PROGRAM OP10_MANUAL
VAR
//OP10A
	OP10A_O_HORZ_MANUALPB1							: BOOL;
	OP10A_O_HORZ_MANUALPB2							: BOOL;
	OP10A_O_VERT_MANUALPB1							: BOOL;
	OP10A_O_VERT_MANUALPB2							: BOOL;
	OP10A_M_O_LHGRIP_ONOFF							: BOOL;
	OP10A_M_O_RHGRIP_ONOFF							: BOOL;
	OP10A_M_O_LHPUSH_CYL							: BOOL;
	OP10A_M_O_RHPUSH_CYL							: BOOL;	
	OP10A_O_0DEGRE_MANUALPB1						: BOOL;
	OP10A_O_180DEGRE_MANUALPB2						: BOOL;
	OP10A_M_LNR1_ONOFF								: BOOL;
	OP10A_M_LNR2_ONOFF								: BOOL;
	OP10A_M_BOWL_ONOFF								: BOOL;
	OP10A_M_HOPPER_ONOFF							: BOOL;
	OP10A_M_LH_REJ_WRK								: BOOL;
	OP10A_M_LH_REJ_HOME								: BOOL;
	OP10A_M_RH_REJ_HOME								: BOOL;
	OP10A_M_RH_REJ_WRK								: BOOL;
	OP10_FRT_BDY_SING_HME							: BOOL;
	OP10_FRT_BDY_SING_WRK							: BOOL;	
	OP10_SEC_BDY_SING_HME							: BOOL;
	OP10_SEC_BDY_SING_WRK							: BOOL;	
	
	
//OP10B                                     		
	OP10B_O_HORZ_MANUALPB1							: BOOL;
	OP10B_O_HORZ_MANUALPB2							: BOOL;
	OP10B_O_VERT_MANUALPB1							: BOOL;
	OP10B_O_VERT_MANUALPB2							: BOOL;
	OP10B_M_O_LHGRIP_ONOFF							: BOOL;
	OP10B_M_O_RHGRIP_ONOFF							: BOOL;
	OP10B_M_O_LHPUSH_CYL							: BOOL;
	OP10B_M_O_RHPUSH_CYL							: BOOL;
	OP10B_O_0DEGRE_MANUALPB1						: BOOL;
	OP10B_O_180DEGRE_MANUALPB2						: BOOL;
	OP10B_M_LNR1_ONOFF								: BOOL;
	OP10B_M_LNR2_ONOFF								: BOOL;
	OP10B_M_BOWL_ONOFF								: BOOL;
	OP10B_M_HOPPER_ONOFF							: BOOL;
	OP10B_M_LH_REJ_HOME								: BOOL;
	OP10B_M_LH_REJ_WRK								: BOOL;
	OP10B_M_RH_REJ_HOME								: BOOL;
	OP10B_M_RH_REJ_WRK								: BOOL;
	
// ALARM BITS

	OP10A_HORZ_CYL_A1								: BOOL;
	OP10A_HORZ_CYL_A2								: BOOL;
	OP10A_HORZ_CYL_A3								: BOOL;
	OP10A_HORZ_CYL_A4								: BOOL;
	OP10A_HORZ_CYL_A5								: BOOL;
	OP10A_VERT_CYL_A1								: BOOL;
	OP10A_VERT_CYL_A2								: BOOL;
	OP10A_VERT_CYL_A3								: BOOL;
	OP10A_VERT_CYL_A4								: BOOL;
	OP10A_VERT_CYL_A5								: BOOL;
	OP10A_DEGREE_CYL_A1								: BOOL;
	OP10A_DEGREE_CYL_A2								: BOOL;
	OP10A_DEGREE_CYL_A3								: BOOL;
	OP10A_DEGREE_CYL_A4								: BOOL;
	OP10A_DEGREE_CYL_A5								: BOOL;
	OP10A_LH_GRP_A1									: BOOL;
	OP10A_LH_GRP_A2									: BOOL;
	OP10A_LH_GRP_A3									: BOOL;
	OP10A_LH_GRP_A4									: BOOL;
	OP10A_LH_GRP_A5									: BOOL;
	OP10A_RH_GRP_A1									: BOOL;
	OP10A_RH_GRP_A2									: BOOL;
	OP10A_RH_GRP_A3									: BOOL;
	OP10A_RH_GRP_A4									: BOOL;
	OP10A_RH_GRP_A5									: BOOL;
	OP10A_LH_PUSH_A1								: BOOL;
	OP10A_LH_PUSH_A2								: BOOL;
	OP10A_LH_PUSH_A3								: BOOL;
	OP10A_LH_PUSH_A4								: BOOL;
	OP10A_LH_PUSH_A5								: BOOL;
	OP10A_RH_PUSH_A1								: BOOL;
	OP10A_RH_PUSH_A2								: BOOL;
	OP10A_RH_PUSH_A3								: BOOL;
	OP10A_RH_PUSH_A4								: BOOL;
	OP10A_RH_PUSH_A5								: BOOL;
	OP10A_LH_REJ_A1									: BOOL;
	OP10A_LH_REJ_A2									: BOOL;
	OP10A_LH_REJ_A3									: BOOL;
	OP10A_LH_REJ_A4									: BOOL;
	OP10A_LH_REJ_A5									: BOOL;
	OP10A_RH_REJ_A1									: BOOL;
	OP10A_RH_REJ_A2									: BOOL;
	OP10A_RH_REJ_A3									: BOOL;
	OP10A_RH_REJ_A4									: BOOL;
	OP10A_RH_REJ_A5									: BOOL;
	OP10B_HORZ_CYL_A1								: BOOL;
	OP10B_HORZ_CYL_A2								: BOOL;
	OP10B_HORZ_CYL_A3								: BOOL;
	OP10B_HORZ_CYL_A4								: BOOL;
	OP10B_HORZ_CYL_A5								: BOOL;
	OP10B_VERT_CYL_A1								: BOOL;
	OP10B_VERT_CYL_A2								: BOOL;
	OP10B_VERT_CYL_A3								: BOOL;
	OP10B_VERT_CYL_A4								: BOOL;
	OP10B_VERT_CYL_A5								: BOOL;
	OP10B_DEGREE_CYL_A1								: BOOL;
	OP10B_DEGREE_CYL_A2								: BOOL;
	OP10B_DEGREE_CYL_A3								: BOOL;
	OP10B_DEGREE_CYL_A4								: BOOL;
	OP10B_DEGREE_CYL_A5								: BOOL;
	OP10B_LH_GRP_A1									: BOOL;
	OP10B_LH_GRP_A2									: BOOL;
	OP10B_LH_GRP_A3									: BOOL;
	OP10B_LH_GRP_A4									: BOOL;
	OP10B_LH_GRP_A5									: BOOL;
	OP10B_RH_GRP_A1									: BOOL;
	OP10B_RH_GRP_A2									: BOOL;
	OP10B_RH_GRP_A3									: BOOL;
	OP10B_RH_GRP_A4									: BOOL;
	OP10B_RH_GRP_A5									: BOOL;
	OP10B_LH_PUSH_A1								: BOOL;
	OP10B_LH_PUSH_A2								: BOOL;
	OP10B_LH_PUSH_A3								: BOOL;
	OP10B_LH_PUSH_A4								: BOOL;
	OP10B_LH_PUSH_A5								: BOOL;
	OP10B_RH_PUSH_A1								: BOOL;
	OP10B_RH_PUSH_A2								: BOOL;
	OP10B_RH_PUSH_A3								: BOOL;
	OP10B_RH_PUSH_A4								: BOOL;
	OP10B_RH_PUSH_A5								: BOOL;
	OP10B_LH_REJ_A1									: BOOL;
	OP10B_LH_REJ_A2									: BOOL;
	OP10B_LH_REJ_A3									: BOOL;
	OP10B_LH_REJ_A4									: BOOL;
	OP10B_LH_REJ_A5									: BOOL;
	OP10B_RH_REJ_A1									: BOOL;
	OP10B_RH_REJ_A2									: BOOL;
	OP10B_RH_REJ_A3									: BOOL;
	OP10B_RH_REJ_A4									: BOOL;
	OP10B_RH_REJ_A5									: BOOL;	
	OP10_BDY_SING_FRT_A1							: BOOL;
	OP10_BDY_SING_FRT_A2							: BOOL;
	OP10_BDY_SING_FRT_A3							: BOOL;
	OP10_BDY_SING_FRT_A4							: BOOL;
	OP10_BDY_SING_FRT_A5							: BOOL;	
	OP10_BDY_SING_SEC_A1							: BOOL;
	OP10_BDY_SING_SEC_A2							: BOOL;
	OP10_BDY_SING_SEC_A3							: BOOL;
	OP10_BDY_SING_SEC_A4							: BOOL;
	OP10_BDY_SING_SEC_A5							: BOOL;	
	
	
	

//INT

	OP10A_HORZ_CYL_STUS								: INT;
	OP10A_VERT_CYL_STUS								: INT;
	OP10A_DEGREE_CYL_STUS							: INT;
	OP10A_LH_GRP_STATS								: INT;
	OP10A_RH_GRP_STUS								: INT;
	OP10A_LH_PUSH_STUS								: INT;
	OP10A_RH_PUSH_STUS								: INT;
	OP10B_HORZ_CYL_STUS								: INT;
	OP10B_VERT_CYL_STUS								: INT;
	OP10B_DEGREE_CYL_STUS							: INT;
	OP10B_LH_GRP_STATS								: INT;
	OP10B_RH_GRP_STUS								: INT;
	OP10B_LH_PUSH_STUS								: INT;
	OP10B_RH_PUSH_STUS								: INT;
                              				
// BOOL                             				
	OP10A_H_LNR1_ONOFF								: BOOL;
	OP10A_H_LNR2_ONOFF								: BOOL;
	OP10A_H_BOWL_ONOFF								: BOOL;
	OP10A_H_HOPPER_ONOFF							: BOOL;
	OP10B_H_LNR1_ONOFF								: BOOL;
	OP10B_H_LNR2_ONOFF								: BOOL;
	OP10B_H_BOWL_ONOFF								: BOOL;
	OP10B_H_HOPPER_ONOFF							: BOOL;

	
	
	
HMI_TRIAL_SWITH_GOKUL_2							:BOOL;	
	
TEMP	: BOOL;
	temp1: BOOL;
	temp2: BOOL;
	OP10_BDY_SING_FRT_STATUS: INT;
	OP10_BDY_SING_SEC_STATUS: INT;




	OP10B_PARLLEL: INT;
	OP10A_PARALLEL: INT;
END_VAR

VAR RETAIN

END_VAR

//#############################		OP10A		###############################

IF OP10A_MANUAL_SELECTED THEN

//OP10A
	OP10A_M_LNR1_ONOFF							:= OP10A_H_LNR1_ONOFF;
	OP10A_M_LNR2_ONOFF          				:= OP10A_H_LNR2_ONOFF;
	OP10A_M_BOWL_ONOFF          				:= OP10A_H_BOWL_ONOFF;
	OP10A_M_HOPPER_ONOFF        				:= OP10A_H_HOPPER_ONOFF;	

CASE OP10_CYL_NO OF                 		
	                                		
	1: IF OP10_HOME THEN            		
		OP10A_O_HORZ_MANUALPB1					:=TRUE;
		OP10A_O_HORZ_MANUALPB2					:=FALSE;
		END_IF                      			
		IF OP10_WORK THEN           			
		OP10A_O_HORZ_MANUALPB1					:=FALSE;
		OP10A_O_HORZ_MANUALPB2					:=TRUE;
		END_IF                      			
                                    			
	2: IF OP10_HOME THEN            			
		OP10A_O_VERT_MANUALPB1					:=TRUE;
		OP10A_O_VERT_MANUALPB2					:=FALSE;
		END_IF                      		
		IF OP10_WORK THEN           		
		OP10A_O_VERT_MANUALPB1					:=FALSE;
		OP10A_O_VERT_MANUALPB2					:=TRUE;
		END_IF                      			
		                            			
	4:IF OP10_HOME THEN             			
		OP10A_O_0DEGRE_MANUALPB1				:=TRUE;
		OP10A_O_180DEGRE_MANUALPB2				:=FALSE;
		END_IF                      			
		IF OP10_WORK THEN           			
		OP10A_O_0DEGRE_MANUALPB1				:=FALSE;
		OP10A_O_180DEGRE_MANUALPB2				:=TRUE;
		END_IF                      		
                            		
	9: IF OP10_HOME THEN            		
		OP10A_M_LH_REJ_HOME						:=TRUE;
		OP10A_M_LH_REJ_WRK		 				:=FALSE;
		END_IF                      			
		IF OP10_WORK THEN           			
		OP10A_M_LH_REJ_HOME						:=FALSE;
		OP10A_M_LH_REJ_WRK	 					:=TRUE;
		END_IF                      			
		                            			
	10: IF OP10_HOME THEN           			
		OP10A_M_RH_REJ_HOME						:=TRUE;
		OP10A_M_RH_REJ_WRK	 	 				:=FALSE;
		END_IF                      			
		IF OP10_WORK THEN           			
		OP10A_M_RH_REJ_HOME						:=FALSE;
		OP10A_M_RH_REJ_WRK	 					:=TRUE;
		END_IF	                    		
		                            		                     		
		                            		
	13: IF OP10_HOME THEN           		
		OP10A_M_O_LHGRIP_ONOFF					:=FALSE;
		END_IF                      			
		IF OP10_WORK THEN           			
		OP10A_M_O_LHGRIP_ONOFF					:=TRUE;
		END_IF                      			
		                            			
	14:	IF OP10_HOME THEN           			
		OP10A_M_O_RHGRIP_ONOFF					:=FALSE;
		END_IF                      			
		IF OP10_WORK THEN           	    	
		OP10A_M_O_RHGRIP_ONOFF					:=TRUE;
		END_IF                      			
		                            			
	15: IF OP10_HOME THEN           			
		OP10A_M_O_LHPUSH_CYL					:=FALSE;
		END_IF                      		
		IF OP10_WORK THEN           		
		OP10A_M_O_LHPUSH_CYL					:=TRUE;
		END_IF                      			
		                            			
	16: IF OP10_HOME THEN           			
		OP10A_M_O_RHPUSH_CYL					:=FALSE;
		END_IF                      			
		IF OP10_WORK THEN           			
		OP10A_M_O_RHPUSH_CYL					:=TRUE;
		END_IF                              	
		                                    	
	17: IF OP10_HOME THEN           			
		OP10_FRT_BDY_SING_HME					:=TRUE;
		OP10_FRT_BDY_SING_WRK 	 				:=FALSE;
		END_IF                      		
		IF OP10_WORK THEN           		
		OP10_FRT_BDY_SING_HME	 				:=FALSE;
		OP10_FRT_BDY_SING_WRK 					:=TRUE;
		END_IF                              	
                                            	
	18: IF OP10_HOME THEN           			
		OP10_SEC_BDY_SING_HME					:=TRUE;
		OP10_SEC_BDY_SING_WRK		 			:=FALSE;
		END_IF                      		
		IF OP10_WORK THEN           		
		OP10_SEC_BDY_SING_HME					:=FALSE;
		OP10_SEC_BDY_SING_WRK					:=TRUE;
		END_IF                              	
                    		                	
		                            	    	
END_CASE

CASE OP10_SERVO_NO OF               	
	                                	
	1: OP10A_SRV_O_CNVY_STUS.jogPos				:= OP10_JOG_POSITIVE AND NOT OP10_JOG_NEGATIVE;
	   OP10A_SRV_O_CNVY_STUS.jogNeg				:= OP10_JOG_NEGATIVE AND NOT OP10_JOG_POSITIVE;
	   OP10A_SRV_O_CNVY_CNT.Bsethome	        := OP10A_SET_HOME;
	   OP10A_SRV_O_CNVY_STUS.targetPositon	    := OP10A_TARGET_POSITION;
	   OP10A_SRV_O_CNVY_STUS.moveAbsolute	    := OP10A_MOVE_TARGET;
	   OP10A_SRV_ACT_POS						:= OP10A_SRV_O_CNVY_STUS.actualPosition;
	   OP10A_SRV_FAULT							:= OP10A_CONVEYOR.bAxisError;
	   OP10A_SRV_ENABLE							:= OP10A_CONVEYOR.bAxisEnabled;

	    
	3: OP10A_SRV_LH_BDYGRP_STUS.jogPos			:= OP10_JOG_POSITIVE AND NOT OP10_JOG_NEGATIVE;
	   OP10A_SRV_LH_BDYGRP_STUS.jogNeg      	:= OP10_JOG_NEGATIVE AND NOT OP10_JOG_POSITIVE;  
	   OP10A_SRV_LH_BDYGRP_CNT.Axis_Home_Cmd	:= OP10A_SET_HOME;
	   OP10A_SRV_LH_BDYGRP_STUS.targetPositon	:= OP10A_TARGET_POSITION;
	   OP10A_SRV_LH_BDYGRP_STUS.moveAbsolute	:= OP10A_MOVE_TARGET;
	   OP10A_SRV_ACT_POS						:= OP10A_SRV_LH_BDYGRP_STUS.actualPosition;
	   OP10A_SRV_FAULT							:= OP10A_LH_GRIPR.bAxisError;
	   OP10A_SRV_ENABLE							:= OP10A_LH_GRIPR.bAxisEnabled;
	   
	4: OP10A_SRV_RH_BDYGRP_STUS.jogPos			:= OP10_JOG_POSITIVE AND NOT OP10_JOG_NEGATIVE;
	   OP10A_SRV_RH_BDYGRP_STUS.jogNeg   		:= OP10_JOG_NEGATIVE AND NOT OP10_JOG_POSITIVE;
	   OP10A_SRV_RH_BDYGRP_CNT.Axis_Home_Cmd	:= OP10A_SET_HOME;
	   OP10A_SRV_RH_BDYGRP_STUS.targetPositon	:= OP10A_TARGET_POSITION;
	   OP10A_SRV_RH_BDYGRP_STUS.moveAbsolute	:= OP10A_MOVE_TARGET;
	   OP10A_SRV_ACT_POS						:= OP10A_SRV_RH_BDYGRP_STUS.actualPosition;
	   OP10A_SRV_FAULT							:= OP10A_RH_GRIPR.bAxisError;
	   OP10A_SRV_ENABLE							:= OP10A_RH_GRIPR.bAxisEnabled;
	                                			
	5: OP10A_SRV_LH_BDYANG_STUS.jogPos			:= OP10_JOG_POSITIVE AND NOT OP10_JOG_NEGATIVE;
	   OP10A_SRV_LH_BDYANG_STUS.jogNeg   		:= OP10_JOG_NEGATIVE AND NOT OP10_JOG_POSITIVE;
	   OP10A_SRV_LH_BDYANG_CNT.Axis_Home_Cmd	:= OP10A_SET_HOME;
	   OP10A_SRV_LH_BDYANG_STUS.targetPositon	:= OP10A_TARGET_POSITION;
	   OP10A_SRV_LH_BDYANG_STUS.moveAbsolute	:= OP10A_MOVE_TARGET;
	   OP10A_SRV_ACT_POS						:= OP10A_SRV_LH_BDYANG_STUS.actualPosition;
	   OP10A_SRV_FAULT							:= OP10A_LH_ROTY.bAxisError;
	   OP10A_SRV_ENABLE							:= OP10A_LH_ROTY.bAxisEnabled;
                                			
	6: OP10A_SRV_RH_BDYANG_STUS.jogPos			:= OP10_JOG_POSITIVE AND NOT OP10_JOG_NEGATIVE;
	   OP10A_SRV_RH_BDYANG_STUS.jogNeg   		:= OP10_JOG_NEGATIVE AND NOT OP10_JOG_POSITIVE;
	   OP10A_SRV_RH_BDYANG_CNT.Axis_Home_Cmd	:= OP10A_SET_HOME;
	   OP10A_SRV_RH_BDYANG_STUS.targetPositon	:= OP10A_TARGET_POSITION;
	   OP10A_SRV_RH_BDYANG_STUS.moveAbsolute	:= OP10A_MOVE_TARGET;
	   OP10A_SRV_ACT_POS						:= OP10A_SRV_RH_BDYANG_STUS.actualPosition;
	   OP10A_SRV_FAULT							:= OP10A_RH_ROTY.bAxisError;
	   OP10A_SRV_ENABLE							:= OP10A_RH_ROTY.bAxisEnabled;
                           			
	11:OP10_SRV_FRST_PCKBDY_STUS.jogPos			:= OP10_JOG_POSITIVE AND NOT OP10_JOG_NEGATIVE;
	   OP10_SRV_FRST_PCKBDY_STUS.jogNeg  		:= OP10_JOG_NEGATIVE AND NOT OP10_JOG_POSITIVE;
	   OP10_SRV_FRST_PCKBDY_CNT.Axis_Home_Cmd	:= OP10A_SET_HOME;
	   OP10_SRV_FRST_PCKBDY_STUS.targetPositon	:= OP10A_TARGET_POSITION;    
	   OP10_SRV_FRST_PCKBDY_STUS.moveAbsolute	:= OP10A_MOVE_TARGET;
	   OP10A_SRV_ACT_POS						:= OP10_SRV_FRST_PCKBDY_STUS.actualPosition;
	   OP10A_SRV_FAULT							:= OP10_FRT_BDY_GPR.bAxisError;
	   OP10A_SRV_ENABLE							:= OP10_FRT_BDY_GPR.bAxisEnabled;

                         			
	12:OP10_SRV_SCND_PCKBDY_STUS.jogPos			:= OP10_JOG_POSITIVE AND NOT OP10_JOG_NEGATIVE;
	   OP10_SRV_SCND_PCKBDY_STUS.jogNeg  		:= OP10_JOG_NEGATIVE AND NOT OP10_JOG_POSITIVE;   
	   OP10_SRV_SCND_PCKBDY_CNT.Axis_Home_Cmd	:= OP10A_SET_HOME;
	   OP10_SRV_SCND_PCKBDY_STUS.targetPositon	:= OP10A_TARGET_POSITION;
	   OP10_SRV_SCND_PCKBDY_STUS.moveAbsolute	:= OP10A_MOVE_TARGET;
	   OP10A_SRV_ACT_POS						:= OP10_SRV_SCND_PCKBDY_STUS.actualPosition;
	   OP10A_SRV_FAULT							:= OP10_SEC_BDY_GPR.bAxisError;
	   OP10A_SRV_ENABLE							:= OP10_SEC_BDY_GPR.bAxisEnabled;	   
END_CASE

ELSE
		OP10_CYL_NO									:=0;	
		OP10A_O_HORZ_MANUALPB1						:=FALSE;
		OP10A_O_HORZ_MANUALPB2						:=FALSE;
		OP10A_O_VERT_MANUALPB1						:=FALSE;
		OP10A_O_VERT_MANUALPB2						:=FALSE;
		OP10A_M_O_LHGRIP_ONOFF						:=FALSE;
		OP10A_O_0DEGRE_MANUALPB1					:=FALSE;
		OP10A_O_180DEGRE_MANUALPB2					:=FALSE;
		OP10A_M_O_LHPUSH_CYL						:=FALSE;
		OP10A_M_LNR1_ONOFF		    				:=FALSE;
		OP10A_M_LNR2_ONOFF          				:=FALSE;
		OP10A_M_BOWL_ONOFF         					:=FALSE;
		OP10A_M_HOPPER_ONOFF       					:=FALSE;
		OP10A_M_O_RHPUSH_CYL						:=FALSE;	
		OP10A_M_O_RHGRIP_ONOFF						:=FALSE;
		OP10A_M_RH_REJ_HOME							:=FALSE;
		OP10A_M_RH_REJ_WRK	 						:=FALSE;
		OP10A_M_LH_REJ_HOME							:=FALSE;
		OP10A_M_LH_REJ_WRK	 						:=FALSE;		
		OP10_FRT_BDY_SING_HME	 					:=FALSE;
		OP10_FRT_BDY_SING_WRK						:=FALSE;
		OP10_SEC_BDY_SING_HME	 					:=FALSE;
		OP10_SEC_BDY_SING_WRK						:=FALSE;		
		
		
		
END_IF
	

//#############################		OP10B		###############################



IF OP10B_MANUAL_SELECTED THEN
//OP10B                         				
	OP10B_M_LNR1_ONOFF          				:= OP10B_H_LNR1_ONOFF  ;
	OP10B_M_LNR2_ONOFF          				:= OP10B_H_LNR2_ONOFF  ;
	OP10B_M_BOWL_ONOFF          				:= OP10B_H_BOWL_ONOFF  ;
	OP10B_M_HOPPER_ONOFF        				:= OP10B_H_HOPPER_ONOFF;	

CASE OP10B_CYL_NO OF 

5: IF OP10B_HOME THEN            		
		OP10B_O_HORZ_MANUALPB1					:=TRUE;
		OP10B_O_HORZ_MANUALPB2					:=FALSE;
		END_IF                      			
		IF OP10B_WORK THEN           			
		OP10B_O_HORZ_MANUALPB1					:=FALSE;
		OP10B_O_HORZ_MANUALPB2					:=TRUE;
		END_IF                      			
                                    			
	6: IF OP10B_HOME THEN            			
		OP10B_O_VERT_MANUALPB1					:=TRUE;
		OP10B_O_VERT_MANUALPB2					:=FALSE;
		END_IF                      			
		IF OP10B_WORK THEN           			
		OP10B_O_VERT_MANUALPB1					:=FALSE;
		OP10B_O_VERT_MANUALPB2					:=TRUE;
		END_IF                      		
		                            		
	8:IF OP10B_HOME THEN             		
		OP10B_O_0DEGRE_MANUALPB1				:=TRUE;
		OP10B_O_180DEGRE_MANUALPB2				:=FALSE;
		END_IF                      			
		IF OP10B_WORK THEN           			
		OP10B_O_0DEGRE_MANUALPB1				:=FALSE;
		OP10B_O_180DEGRE_MANUALPB2				:=TRUE;
		END_IF                              	
	                                        	
	11: IF OP10B_HOME THEN           			
		OP10B_M_LH_REJ_HOME						:=TRUE;
		OP10B_M_LH_REJ_WRK	 	 				:=FALSE;
		END_IF                      		
		IF OP10B_WORK THEN           		
		OP10B_M_LH_REJ_HOME						:=FALSE;
		OP10B_M_LH_REJ_WRK	 					:=TRUE;
		END_IF                      			
                       			            	
	12: IF OP10B_HOME THEN           			
		OP10B_M_RH_REJ_HOME						:=TRUE;
		OP10B_M_RH_REJ_WRK	  	 				:=FALSE;
		END_IF                      			
		IF OP10B_WORK THEN           			
		OP10B_M_RH_REJ_HOME						:=FALSE;
		OP10B_M_RH_REJ_WRK	 					:=TRUE;
		END_IF 	

	17: IF OP10B_HOME THEN           		
		OP10B_M_O_LHGRIP_ONOFF					:=FALSE;
		END_IF                      			
		IF OP10B_WORK THEN           			
		OP10B_M_O_LHGRIP_ONOFF					:=TRUE;
		END_IF                      			
		                            			
	18:	IF OP10B_HOME THEN           			
		OP10B_M_O_RHGRIP_ONOFF					:=FALSE;
		END_IF                      			
		IF OP10B_WORK THEN           			
		OP10B_M_O_RHGRIP_ONOFF					:=TRUE;
		END_IF                      			
		                            			
	19: IF OP10B_HOME THEN           			
		OP10B_M_O_LHPUSH_CYL					:=FALSE;
		END_IF                      		
		IF OP10B_WORK THEN           		
		OP10B_M_O_LHPUSH_CYL					:=TRUE;
		END_IF                      			
		                            			
	20: IF OP10B_HOME THEN           			
		OP10B_M_O_RHPUSH_CYL					:=FALSE;
		END_IF                      			
		IF OP10B_WORK THEN           			
		OP10B_M_O_RHPUSH_CYL					:=TRUE;
		END_IF 

END_CASE	
	
CASE OP10B_SERVO_NO OF 
	
	2: OP10B_SRV_O_CNVY_STUS.jogPos				:= OP10B_JOG_POSITIVE AND NOT OP10B_JOG_NEGATIVE;
	   OP10B_SRV_O_CNVY_STUS.jogNeg				:= OP10B_JOG_NEGATIVE AND NOT OP10B_JOG_POSITIVE;
	   OP10B_SRV_O_CNVY_CNT.Bsethome	        := OP10B_SET_HOME;
	   OP10B_SRV_O_CNVY_STUS.targetPositon	    := OP10B_TARGET_POSITION;
//	   OP10B_SRV_LH_BDYGRP_STUS.targetVelocity	:= OP10B_TARGET_VEL;
	   OP10B_SRV_O_CNVY_STUS.moveAbsolute	    := OP10B_MOVE_TARGET;
	   OP10B_SRV_ACT_POS						:= OP10B_SRV_O_CNVY_STUS.actualPosition;
	   OP10B_SRV_FAULT							:= OP10B_CONVEYOR.bAxisError;
	   OP10B_SRV_ENABLE							:= OP10B_CONVEYOR.bAxisEnabled;
                                    	
	7: OP10B_SRV_LH_BDYGRP_STUS.jogPos			:= OP10B_JOG_POSITIVE AND NOT OP10B_JOG_NEGATIVE;
	   OP10B_SRV_LH_BDYGRP_STUS.jogNeg			:= OP10B_JOG_NEGATIVE AND NOT OP10B_JOG_POSITIVE;
	   OP10B_SRV_LH_BDYGRP_CNT.Axis_Home_Cmd	:= OP10B_SET_HOME;
	   OP10B_SRV_LH_BDYGRP_STUS.targetPositon	:= OP10B_TARGET_POSITION;
//	   OP10B_SRV_LH_BDYGRP_STUS.targetVelocity	:= OP10B_TARGET_VEL;
	   OP10B_SRV_LH_BDYGRP_STUS.moveAbsolute	:= OP10B_MOVE_TARGET;
	   OP10B_SRV_ACT_POS						:= OP10B_SRV_LH_BDYGRP_STUS.actualPosition;
	   OP10B_SRV_FAULT							:= OP10B_LH_GRIPR.bAxisError;
	   OP10B_SRV_ENABLE							:= OP10B_LH_GRIPR.bAxisEnabled;	   
	   
	                                		
	8: OP10B_SRV_RH_BDYGRP_STUS.jogPos			:= OP10B_JOG_POSITIVE AND NOT OP10B_JOG_NEGATIVE;
	   OP10B_SRV_RH_BDYGRP_STUS.jogNeg    		:= OP10B_JOG_NEGATIVE AND NOT OP10B_JOG_POSITIVE;
	   OP10B_SRV_RH_BDYGRP_CNT.Axis_Home_Cmd	:= OP10B_SET_HOME;
	   OP10B_SRV_RH_BDYGRP_STUS.targetPositon	:= OP10B_TARGET_POSITION;
//	   OP10B_SRV_RH_BDYGRP_STUS.targetVelocity	:= OP10B_TARGET_VEL;
	   OP10B_SRV_RH_BDYGRP_STUS.moveAbsolute	:= OP10B_MOVE_TARGET;
	   OP10B_SRV_ACT_POS						:= OP10B_SRV_RH_BDYGRP_STUS.actualPosition;
	   OP10B_SRV_FAULT							:= OP10B_RH_GRIPR.bAxisError;
	   OP10B_SRV_ENABLE							:= OP10B_RH_GRIPR.bAxisEnabled;	
	   
	                                			
	9: OP10B_SRV_LH_BDYANG_STUS.jogPos			:= OP10B_JOG_POSITIVE AND NOT OP10B_JOG_NEGATIVE;
	   OP10B_SRV_LH_BDYANG_STUS.jogNeg   		:= OP10B_JOG_NEGATIVE AND NOT OP10B_JOG_POSITIVE;
	   OP10B_SRV_LH_BDYANG_CNT.Axis_Home_Cmd	:= OP10B_SET_HOME;
	   OP10B_SRV_LH_BDYANG_STUS.targetPositon	:= OP10B_TARGET_POSITION;
//	   OP10B_SRV_LH_BDYANG_STUS.targetVelocity	:= OP10B_TARGET_VEL;
	   OP10B_SRV_LH_BDYANG_STUS.moveAbsolute	:= OP10B_MOVE_TARGET;
	   OP10B_SRV_ACT_POS						:= OP10B_SRV_LH_BDYANG_STUS.actualPosition;
	   OP10B_SRV_FAULT							:= OP10B_LH_ROTY.bAxisError;
	   OP10B_SRV_ENABLE							:= OP10B_LH_ROTY.bAxisEnabled;	   
	                                			
	10:OP10B_SRV_RH_BDYANG_STUS.jogPos			:= OP10B_JOG_POSITIVE AND NOT OP10B_JOG_NEGATIVE;
	   OP10B_SRV_RH_BDYANG_STUS.jogNeg    		:= OP10B_JOG_NEGATIVE AND NOT OP10B_JOG_POSITIVE;
	   OP10B_SRV_RH_BDYANG_CNT.Axis_Home_Cmd	:= OP10B_SET_HOME;
	   OP10B_SRV_RH_BDYANG_STUS.targetPositon	:= OP10B_TARGET_POSITION;
//	   OP10B_SRV_RH_BDYANG_STUS.targetVelocity	:= OP10B_TARGET_VEL;
	   OP10B_SRV_RH_BDYANG_STUS.moveAbsolute	:= OP10B_MOVE_TARGET;
	   OP10B_SRV_ACT_POS						:= OP10B_SRV_RH_BDYANG_STUS.actualPosition;
	   OP10B_SRV_FAULT							:= OP10B_RH_ROTY.bAxisError;
	   OP10B_SRV_ENABLE							:= OP10B_RH_ROTY.bAxisEnabled;	

END_CASE	

ELSE
	OP10B_O_HORZ_MANUALPB1						:=FALSE;		
	OP10B_O_HORZ_MANUALPB2						:=FALSE;		
	OP10B_O_VERT_MANUALPB1						:=FALSE;		
	OP10B_O_VERT_MANUALPB2						:=FALSE;		
	OP10B_M_O_LHGRIP_ONOFF						:=FALSE;		
	OP10B_O_0DEGRE_MANUALPB1					:=FALSE;	
	OP10B_O_180DEGRE_MANUALPB2					:=FALSE;
	OP10B_M_O_LHPUSH_CYL  						:=FALSE;		
	OP10B_M_LNR1_ONOFF  						:=FALSE;		
	OP10B_M_LNR2_ONOFF  						:=FALSE;		
	OP10B_M_BOWL_ONOFF  						:=FALSE;		
	OP10B_M_O_RHPUSH_CYL						:=FALSE;
	OP10B_M_O_RHGRIP_ONOFF						:=FALSE;	
	OP10B_M_RH_REJ_HOME							:=FALSE;
	OP10B_M_RH_REJ_WRK	  	 					:=FALSE;	
	OP10B_M_LH_REJ_HOME							:=FALSE;
	OP10B_M_LH_REJ_WRK	 						:=FALSE;

END_IF
// OP10B_HORZ_CYLINDER_SAFE_WRK/HME
OP10A_HORZ_CYL.SafeHome				:=OP10A_VERT_CYL.Sensor1 ;//AND OP10A_DEGREE_CYL.Sensor1;
OP10A_HORZ_CYL.SafeWork             :=OP10A_VERT_CYL.Sensor1 ;//AND OP10A_DEGREE_CYL.Sensor1;


OP10A_HORZ_CYL(
	Auto:= OP10A_AUTO_RUNNING OR OP10A_STEP_RUNNING OR OP10A_CYL_PNP_CHECK, 
	Manual:= OP10A_MANUAL_SELECTED,
	HOMING_RUNNING:= OP10A_START_HOMNG, 
	ErrorActive:= OP10A_ERR, 
	ResetPB:= Servo_Reset, 								
	Sensor1:= I10A_ORING_HORZ_CYL_REV_I1011_2,         						(*OP10A_HORZ_CYL_FUNTIONAL_BLCK*)                                
	Sensor2:= I10A_ORING_HORZ_CYL_FWD_I1011_3, 
	ManualPB1:= OP10A_O_HORZ_MANUALPB1, 
	ManualPB2:= OP10A_O_HORZ_MANUALPB2, 
	AutoCmd1:= OP10A_O_HORZ_AUTOCMD1, 
	AutoCmd2:= OP10A_O_HORZ_AUTOCMD2, 
	OperationEnable:= OperationEnable, 
	SafeHome:= , 
	SafeWork:= , 
	Pulse_1Sec:= Pulse_Block.Q1Hz, 
	BlinkingBit:= , 
	TimeOut1:= 5, 
	TimeOut2:= 5, 
	TimeOut3:= 5,
	HOMING_STRT:= (OP10A_HME_STP_NO=15), 
	HME_DLY:= 100, 
	HME_DN_NO:= OP10A_HME_15_20, 
	HME_CYL_2:= TRUE, 
	HME_CYL_3:= TRUE, 
	Solenoid1=> O10A_ORING_HORZ_CYL_REV_Q1050_6, 
	Solenoid2=> O10A_ORING_HORZ_CYL_FWD_Q1050_7, 
	AlarmSensor1=> OP10A_HORZ_CYL_A1, 
	AlarmSensor2=> OP10A_HORZ_CYL_A2, 
	AlarmSolenoid1=> OP10A_HORZ_CYL_A3, 
	AlarmSolenoid2=> OP10A_HORZ_CYL_A4, 
	AllSignal=> OP10A_HORZ_CYL_A5, 
	AlarmPresent=> OP10A_CYLINDER_ERR.0, 
	Position1=> , 
	Position2=> , 
	HomeSensorBlink=> , 
	WorkSensorBlink=> ,
	Status:= OP10A_HORZ_CYL_STUS,
	HMENG_RESULT := OP10A_HME_STP_NO);
	

// OP10A_VERT_CYLINDER_SAFE_WRK/HME
OP10A_VERT_CYL.SafeHome				:= OP10A_HORZ_CYL.Sensor1 OR OP10A_HORZ_CYL.Sensor2;
OP10A_VERT_CYL.SafeWork				:= (OP10A_HORZ_CYL.Sensor1 OR OP10A_HORZ_CYL.Sensor2) AND OP10A_DEGREE_CYL.Sensor1;
	
OP10A_VERT_CYL(
	Auto:= OP10A_AUTO_RUNNING OR OP10A_STEP_RUNNING OR OP10A_CYL_PNP_CHECK, 
	Manual:= OP10A_MANUAL_SELECTED,
	HOMING_RUNNING:= OP10A_START_HOMNG, 
	ErrorActive:= OP10A_ERR, 
	ResetPB:= Servo_Reset, 
	Sensor1:= I10A_ORING_VERT_CYL_UP_I1011_4, 
	Sensor2:= I10A_ORING_VERT_CYL_DWN_I1011_5, 								(*OP10A_VERT_CYL_FUNTIONAL_BLOCK*)
	ManualPB1:= OP10A_O_VERT_MANUALPB1, 
	ManualPB2:= OP10A_O_VERT_MANUALPB2, 
	AutoCmd1:= OP10A_O_VERT_AUTOCMD1, 
	AutoCmd2:= OP10A_O_VERT_AUTOCMD2, 
	OperationEnable:= OperationEnable, 
	SafeHome:= , 
	SafeWork:= , 
	Pulse_1Sec:= Pulse_Block.Q1Hz, 
	BlinkingBit:= , 
	TimeOut1:= 5, 
	TimeOut2:= 5, 
	TimeOut3:= 5,
	HOMING_STRT:= (OP10A_HME_STP_NO=20), 
	HME_DLY:= 100, 
	HME_DN_NO:= OP10A_HME_20_25, 
	HME_CYL_2:=TRUE , 
	HME_CYL_3:=TRUE , 
	Solenoid1=> O10A_ORING_VERT_CYL_UP_Q1051_0, 
	Solenoid2=> O10A_ORING_VERT_CYL_DWN_Q1051_1, 
	AlarmSensor1=> OP10A_VERT_CYL_A1, 
	AlarmSensor2=> OP10A_VERT_CYL_A2, 
	AlarmSolenoid1=> OP10A_VERT_CYL_A3, 
	AlarmSolenoid2=> OP10A_VERT_CYL_A4, 
	AllSignal=> OP10A_VERT_CYL_A5, 
	AlarmPresent=> OP10A_CYLINDER_ERR.1, 
	Position1=> , 
	Position2=> , 
	HomeSensorBlink=> , 
	WorkSensorBlink=> ,
	Status:= OP10A_VERT_CYL_STUS,
	HMENG_RESULT := OP10A_HME_STP_NO);

// OP10A_DEGREE_CYLINDER_SAFE_WRK/HME	
OP10A_DEGREE_CYL.SafeHome				:= OP10A_HORZ_CYL.Sensor1 AND OP10A_VERT_CYL.Sensor1;
OP10A_DEGREE_CYL.SafeWork				:= OP10A_HORZ_CYL.Sensor1 AND OP10A_VERT_CYL.Sensor1; 
	
	
OP10A_DEGREE_CYL(
	Auto:= OP10A_AUTO_RUNNING OR OP10A_STEP_RUNNING OR OP10A_CYL_PNP_CHECK, 
	Manual:= OP10A_MANUAL_SELECTED,
	HOMING_RUNNING:= OP10A_START_HOMNG, 
	ErrorActive:= OP10A_ERR, 
	ResetPB:= Servo_Reset, 
	Sensor1:= I10A_ORING_ROTRY_CYL_O_DEG_I1011_0, 							(*OP10A_DEGREE_CYL_FUNTIONAL_BLCK*)
	Sensor2:= I10A_ORING_ROTRY_CYL_180_DEG_I1011_1, 
	ManualPB1:= OP10A_O_0DEGRE_MANUALPB1, 
	ManualPB2:= OP10A_O_180DEGRE_MANUALPB2, 
	AutoCmd1:= OP10A_O_0DEGRE_AUTOCMD1, 
	AutoCmd2:= OP10A_O_180DEGRE_AUTOCMD2, 
	OperationEnable:= OperationEnable, 
	SafeHome:= , 
	SafeWork:= , 
	Pulse_1Sec:= Pulse_Block.Q1Hz, 
	BlinkingBit:= , 
	TimeOut1:= 5, 
	TimeOut2:= 5, 
	TimeOut3:= 5,
	HOMING_STRT:= (OP10A_HME_STP_NO=25), 
	HME_DLY:= 100, 
	HME_DN_NO:=  OP10A_HME_25_30, 
	HME_CYL_2:=TRUE , 
	HME_CYL_3:=TRUE , 
	Solenoid1=> O10A_ORING_ROTRY_CYL_O_DEG_Q1050_4, 
	Solenoid2=> O10A_ORING_ROTRY_CYL_180_DEG_Q1050_5, 
	AlarmSensor1=> OP10A_DEGREE_CYL_A1, 
	AlarmSensor2=> OP10A_DEGREE_CYL_A2, 
	AlarmSolenoid1=> OP10A_DEGREE_CYL_A3, 
	AlarmSolenoid2=> OP10A_DEGREE_CYL_A4, 
	AllSignal=> OP10A_DEGREE_CYL_A5, 
	AlarmPresent=> OP10A_CYLINDER_ERR.2, 
	Position1=> , 
	Position2=> , 
	HomeSensorBlink=> , 
	WorkSensorBlink=> ,
	Status:= OP10A_DEGREE_CYL_STUS,
	HMENG_RESULT := OP10A_HME_STP_NO);
	
// OP10A_LH_GRIPPER_CYLINDER_SAFE_WRK/HME	
OP10A_LH_GRP.SafeHome						:= OP10A_LH_PUSH.Sensor1;
OP10A_LH_GRP.SafeWork						:= OP10A_LH_PUSH.Sensor1;

	
OP10A_LH_GRP(
	Auto:= OP10A_AUTO_RUNNING OR OP10A_STEP_RUNNING OR OP10A_CYL_PNP_CHECK, 
	Manual:= OP10A_MANUAL_SELECTED,
	HOMING_RUNNING:= OP10A_START_HOMNG, 
	ErrorActive:= OP10A_ERR, 
	ResetPB:= Servo_Reset, 
	Sensor1:= I10A_ORING_LH_GRPR_CLSE_I1010_2, 								(*OP10A_LH_GRIPPER_FUNCATIONAL_BLOCK*)
	Sensor2:= I10A_ORING_LH_GRPR_OPN_I1010_3, 
	ManualPB1:=OP10A_LH_GRP.Manual AND  NOT OP10A_M_O_LHGRIP_ONOFF,//NOT OP10A_M_O_LHGRIP_ONOFF, 
	ManualPB2:=OP10A_LH_GRP.Manual AND OP10A_M_O_LHGRIP_ONOFF,//OP10A_M_O_LHGRIP_ONOFF, 
	AutoCmd1:=OP10A_LH_GRP.Auto AND NOT OP10A_A_O_LHGRIP_ONOFF,// NOT OP10A_A_O_LHGRIP_ONOFF, 
	AutoCmd2:=OP10A_LH_GRP.Auto AND OP10A_A_O_LHGRIP_ONOFF, 
	OperationEnable:= OperationEnable, 
	SafeHome:= 1, 
	SafeWork:= 1, 
	Pulse_1Sec:= Pulse_Block.Q1Hz, 
	BlinkingBit:= , 
	TimeOut1:= 5, 
	TimeOut2:= 5, 
	TimeOut3:= 5,
	HOMING_STRT:=(OP10A_HME_STP_NO=5), 
	HME_DLY:= 100, 
	HME_DN_NO:= OP10A_HME_5_10, 
	HME_CYL_2:= OP10A_RH_GRP.Sensor1, 
	HME_CYL_3:=TRUE , 
	Solenoid1=> , 
	Solenoid2=>O10A_ORING_LH_GRPR_CLSE_OPN_Q1050_0 , 
	AlarmSensor1=> OP10A_LH_GRP_A1, 
	AlarmSensor2=> OP10A_LH_GRP_A2, 
	AlarmSolenoid1=> OP10A_LH_GRP_A3, 
	AlarmSolenoid2=> OP10A_LH_GRP_A4, 
	AllSignal=> OP10A_LH_GRP_A5, 
	AlarmPresent=> OP10A_CYLINDER_ERR.3, 
	Position1=> , 
	Position2=> , 
	HomeSensorBlink=> , 
	WorkSensorBlink=> ,	
	Status:= OP10A_LH_GRP_STATS,
	HMENG_RESULT := OP10A_HME_STP_NO);

// OP10A_RH_GRIPPER_CYLINDER_SAFE_WRK/HME	
OP10A_RH_GRP.SafeHome						:= OP10A_RH_PUSH.Sensor1;
OP10A_RH_GRP.SafeWork						:= OP10A_RH_PUSH.Sensor1;				// CHANGE THE INPUT AS FALSE

	
	
OP10A_RH_GRP(
	Auto:= OP10A_AUTO_RUNNING OR OP10A_STEP_RUNNING OR OP10A_CYL_PNP_CHECK, 
	Manual:= OP10A_MANUAL_SELECTED,
	HOMING_RUNNING:= OP10A_START_HOMNG, 
	ErrorActive:= OP10A_ERR, 
	ResetPB:= Servo_Reset, 
	Sensor1:= I10A_ORING_RH_GRPR_CLSE_I1010_6, 
	Sensor2:= I10A_ORING_RH_GRPR_OPN_I1010_5, 
	ManualPB1:=OP10A_RH_GRP.Manual AND  NOT OP10A_M_O_RHGRIP_ONOFF, 
	ManualPB2:= OP10A_RH_GRP.Manual AND OP10A_M_O_RHGRIP_ONOFF, 									(*OP10A_RH_GRIPPER_CYLINDER*)
	AutoCmd1:=OP10A_RH_GRP.Auto AND NOT OP10A_A_O_RHGRIP_ONOFF, 
	AutoCmd2:=OP10A_RH_GRP.Auto AND OP10A_A_O_RHGRIP_ONOFF, 
	OperationEnable:= OperationEnable, 
	SafeHome:= 1, 
	SafeWork:= 1, 
	Pulse_1Sec:= Pulse_Block.Q1Hz, 
	BlinkingBit:= , 
	TimeOut1:= 5, 
	TimeOut2:= 5, 
	TimeOut3:= 5,
	HOMING_STRT:= (OP10A_HME_STP_NO=5),
	HME_DLY:= ,
	HME_DN_NO:= ,
	HME_CYL_2:=TRUE ,
	HME_CYL_3:=TRUE , 
	Solenoid1=> , 
	Solenoid2=> O10A_ORING_RH_GRPR_CLSE_OPN_Q1050_2, 
	AlarmSensor1=> OP10A_RH_GRP_A1, 
	AlarmSensor2=> OP10A_RH_GRP_A2, 
	AlarmSolenoid1=> OP10A_RH_GRP_A3, 
	AlarmSolenoid2=> OP10A_RH_GRP_A4, 
	AllSignal=> OP10A_RH_GRP_A5, 
	AlarmPresent=> OP10A_CYLINDER_ERR.4, 
	Position1=> , 
	Position2=> , 
	HomeSensorBlink=> , 
	WorkSensorBlink=> ,	
	Status:= OP10A_RH_GRP_STUS,
	HMENG_RESULT := OP10A_PARALLEL);

// OP10A_LH_PUSH_CYLINDER_SAFE_WRK/HME
OP10A_LH_PUSH.SafeHome						:=OP10A_LH_GRP.Sensor2 ;
OP10A_LH_PUSH.SafeWork						:=OP10A_LH_GRP.Sensor2 ;

	
OP10A_LH_PUSH(
	Auto:= OP10A_AUTO_RUNNING OR OP10A_STEP_RUNNING OR OP10A_CYL_PNP_CHECK, 
	Manual:= OP10A_MANUAL_SELECTED,
	HOMING_RUNNING:= OP10A_START_HOMNG, 
	ErrorActive:= OP10A_ERR, 
	ResetPB:= Servo_Reset, 
	Sensor1:= NOT I10A_ORING_LH_PUSHR_CYL_REV_I1010_4, 										(*OP10A_LH_PUSHING_CYLINDER*)
	Sensor2:= I10A_ORING_LH_PUSHR_CYL_REV_I1010_4, 
	ManualPB1:=OP10A_LH_PUSH.Manual AND NOT OP10A_M_O_LHPUSH_CYL, 
	ManualPB2:=OP10A_LH_PUSH.Manual AND OP10A_M_O_LHPUSH_CYL, 
	AutoCmd1:=OP10A_LH_PUSH.Auto AND NOT OP10A_A_O_LHPUSH_CYL, 
	AutoCmd2:=OP10A_LH_PUSH.Auto AND OP10A_A_O_LHPUSH_CYL, 
	OperationEnable:= OperationEnable, 
	SafeHome:= , 
	SafeWork:= , 
	Pulse_1Sec:= Pulse_Block.Q1Hz, 
	BlinkingBit:= , 
	TimeOut1:= 5, 
	TimeOut2:= 5, 
	TimeOut3:= 5,
	HOMING_STRT:= (OP10A_HME_STP_NO=1),
	HME_DLY:= 100,
	HME_DN_NO:= OP10A_HME_1_5,
	HME_CYL_2:= OP10A_RH_PUSH.Sensor1,
	HME_CYL_3:=TRUE , 
	Solenoid1=> , 
	Solenoid2=> O10A_ORING_LH_PUSHR_CYL_REV_FWD_Q1050_1, 
	AlarmSensor1=> OP10A_LH_PUSH_A1, 
	AlarmSensor2=> OP10A_LH_PUSH_A2, 
	AlarmSolenoid1=> OP10A_LH_PUSH_A3, 
	AlarmSolenoid2=> OP10A_LH_PUSH_A4, 
	AllSignal=> OP10A_LH_PUSH_A5, 
	AlarmPresent=> OP10A_CYLINDER_ERR.5, 
	Position1=> , 
	Position2=> , 
	HomeSensorBlink=> , 
	WorkSensorBlink=> ,	
	Status:= OP10A_LH_PUSH_STUS,
	HMENG_RESULT := OP10A_HME_STP_NO);


// OP10A_LH_PUSH_CYLINDER_SAFE_WRK/HME
OP10A_RH_PUSH.SafeHome						:= OP10A_RH_GRP.Sensor2 ;
OP10A_RH_PUSH.SafeWork						:= OP10A_RH_GRP.Sensor2 ;


OP10A_RH_PUSH(
	Auto:= OP10A_AUTO_RUNNING OR OP10A_STEP_RUNNING OR OP10A_CYL_PNP_CHECK, 
	Manual:= OP10A_MANUAL_SELECTED,
	HOMING_RUNNING:= OP10A_START_HOMNG, 
	ErrorActive:= OP10A_ERR, 								(*OP10A_RH _ PUSHING CYL_FUNTIONAL_BLCK*)
	ResetPB:= Servo_Reset, 
	Sensor1:= NOT I10A_ORING_RH_PUSHR_CYL_REV_I1010_7, 
	Sensor2:=I10A_ORING_RH_PUSHR_CYL_REV_I1010_7 , 
	ManualPB1:=OP10A_RH_PUSH.Manual AND NOT OP10A_M_O_RHPUSH_CYL, 
	ManualPB2:=OP10A_RH_PUSH.Manual AND OP10A_M_O_RHPUSH_CYL, 
	AutoCmd1:=OP10A_RH_PUSH.AUTO AND NOT OP10A_A_O_RHPUSH_CYL, 
	AutoCmd2:= OP10A_RH_PUSH.AUTO AND OP10A_A_O_RHPUSH_CYL, 
	OperationEnable:= OperationEnable, 
	SafeHome:= , 
	SafeWork:= , 
	Pulse_1Sec:= Pulse_Block.Q1Hz, 
	BlinkingBit:= , 
	TimeOut1:= 5, 
	TimeOut2:= 5, 
	TimeOut3:= 5,
	HOMING_STRT:= (OP10A_HME_STP_NO=1),
	HME_DLY:= ,
	HME_DN_NO:= ,
	HME_CYL_2:=TRUE ,
	HME_CYL_3:=TRUE , 
	Solenoid1=> , 
	Solenoid2=>O10A_ORING_RH_PUSHR_CYL_REV_FWD_Q1050_3 , 
	AlarmSensor1=> OP10A_RH_PUSH_A1, 
	AlarmSensor2=> OP10A_RH_PUSH_A2, 
	AlarmSolenoid1=> OP10A_RH_PUSH_A3, 
	AlarmSolenoid2=> OP10A_RH_PUSH_A4, 
	AllSignal=> OP10A_RH_PUSH_A5, 
	AlarmPresent=> OP10A_CYLINDER_ERR.6, 
	Position1=> , 
	Position2=> , 
	HomeSensorBlink=> , 
	WorkSensorBlink=> ,	
	Status:= OP10A_RH_PUSH_STUS,
	HMENG_RESULT := OP10A_PARALLEL);
	
// OP10A_LH_REJ_CYLINDER_SAFE_WRK/HME
//OP10A_LH_REJ.SafeHome						:= TRUE;
//OP10A_LH_REJ.SafeWork						:= TRUE;

OP10A_LH_REJ(
	Auto:= OP10A_AUTO_RUNNING OR OP10A_STEP_RUNNING OR OP10A_CYL_PNP_CHECK, 
	Manual:= OP10A_MANUAL_SELECTED,
	HOMING_RUNNING:= OP10A_START_HOMNG, 
	ErrorActive:= OP10A_ERR, 								(*OP10A_RH _ PUSHING CYL_FUNTIONAL_BLCK*)
	ResetPB:= Servo_Reset, 
	Sensor1:= I10A_LH_FIRTRE_ORING_REJ_CYL_REV_I1011_6, 
	Sensor2:= I10A_LH_FIRTRE_ORING_REJ_CYL_FWD_I1011_7 , 
	ManualPB1:= OP10A_M_LH_REJ_HOME, 
	ManualPB2:= OP10A_M_LH_REJ_WRK, 
	AutoCmd1:= OP10A_A_LH_REJ_HOME, 
	AutoCmd2:= OP10A_A_LH_REJ_WRK, 
	OperationEnable:= OperationEnable, 
	SafeHome:= 1, 
	SafeWork:= 1, 
	Pulse_1Sec:= Pulse_Block.Q1Hz, 
	BlinkingBit:= , 
	TimeOut1:= 5, 
	TimeOut2:= 5, 
	TimeOut3:= 5,
	HOMING_STRT:= (OP10A_HME_STP_NO=1),
	HME_DLY:= ,
	HME_DN_NO:= ,
	HME_CYL_2:=TRUE ,
	HME_CYL_3:=TRUE , 
	Solenoid1=>O10A_LH_FIRTRE_ORING_REJ_CYL_REV_Q1051_2 , 
	Solenoid2=>O10A_LH_FIRTRE_ORING_REJ_CYL_FWD_Q1051_3 , 						
	AlarmSensor1=> OP10A_LH_REJ_A1,                    
	AlarmSensor2=> OP10A_LH_REJ_A2,                    
	AlarmSolenoid1=>OP10A_LH_REJ_A3,                   
	AlarmSolenoid2=> OP10A_LH_REJ_A4, 
	AllSignal=> OP10A_LH_REJ_A5, 
	AlarmPresent=> OP10A_CYLINDER_ERR.7, 
	Position1=> , 
	Position2=> , 
	HomeSensorBlink=> , 
	WorkSensorBlink=> ,	
	Status:= OP10A_RH_PUSH_STUS,
	HMENG_RESULT := OP10A_PARALLEL);	
	
// OP10A_RH_REJ_CYLINDER_SAFE_WRK/HME
//OP10A_RH_REJ.SafeHome						:= TRUE;
//OP10A_RH_REJ.SafeWork						:= TRUE;

OP10A_RH_REJ(
	Auto:= OP10A_AUTO_RUNNING OR OP10A_STEP_RUNNING OR OP10A_CYL_PNP_CHECK, 
	Manual:= OP10A_MANUAL_SELECTED,
	HOMING_RUNNING:= OP10A_START_HOMNG, 
	ErrorActive:= OP10A_ERR, 								(*OP10A_RH _ PUSHING CYL_FUNTIONAL_BLCK*)
	ResetPB:= Servo_Reset, 
	Sensor1:= I10A_RH_FIRTRE_ORING_REJ_CYL_REV_I1020_0, 
	Sensor2:= I10A_RH_FIRTRE_ORING_REJ_CYL_FWD_I1020_1, 
	ManualPB1:= OP10A_M_RH_REJ_HOME, 
	ManualPB2:= OP10A_M_RH_REJ_WRK, 
	AutoCmd1:= OP10A_A_RH_REJ_HOME, 
	AutoCmd2:= OP10A_A_RH_REJ_WRK, 
	OperationEnable:= OperationEnable, 
	SafeHome:= 1, 
	SafeWork:= 1, 
	Pulse_1Sec:= Pulse_Block.Q1Hz, 
	BlinkingBit:= , 
	TimeOut1:= 5, 
	TimeOut2:= 5, 
	TimeOut3:= 5,
	HOMING_STRT:= (OP10A_HME_STP_NO=1),
	HME_DLY:= ,
	HME_DN_NO:= ,
	HME_CYL_2:=TRUE ,
	HME_CYL_3:=TRUE , 
	Solenoid1=>O10A_RH_FIRTRE_ORING_REJ_CYL_REV_Q1051_4 , 
	Solenoid2=>O10A_RH_FIRTRE_ORING_REJ_CYL_FWD_Q1051_5 , 
	AlarmSensor1=>  OP10A_RH_REJ_A1,	
	AlarmSensor2=>  OP10A_RH_REJ_A2,	
	AlarmSolenoid1=>OP10A_RH_REJ_A3,	 
	AlarmSolenoid2=> OP10A_RH_REJ_A4, 
	AllSignal=>  OP10A_RH_REJ_A5,	
	AlarmPresent=> OP10A_CYLINDER_ERR.8, 
	Position1=> , 
	Position2=> , 
	HomeSensorBlink=> , 
	WorkSensorBlink=> ,	
	Status:= OP10A_RH_PUSH_STUS,
	HMENG_RESULT := OP10A_PARALLEL);	




////////////////////////////////////OP10B_CYLINDER_BLOCK////////////////////////////////////
// OP10B_HORZ_CYLINDER_SAFE_WRK/HME
OP10B_HORZ_CYL.SafeHome				:=OP10B_VERT_CYL.Sensor1 ;//AND OP10B_DEGREE_CYL.Sensor1;
OP10B_HORZ_CYL.SafeWork             :=OP10B_VERT_CYL.Sensor1 ;//AND OP10B_DEGREE_CYL.Sensor1;

OP10B_HORZ_CYL(
	Auto:= OP10B_AUTO_RUNNING OR OP10B_STEP_RUNNING OR OP10B_CYL_PNP_CHECK , 
	Manual:= OP10B_MANUAL_SELECTED,
	HOMING_RUNNING:= OP10B_START_HOMNG, 
	ErrorActive:= OP10B_ERR, 
	ResetPB:= Servo_Reset, 								
	Sensor1:= I10B_ORING_HORZ_CYL_REV_I1031_2,         						(*OP10B_HORZ_CYL_FUNTIONAL_BLCK*)                                
	Sensor2:= I10B_ORING_HORZ_CYL_FWD_I1031_3, 
	ManualPB1:= OP10B_O_HORZ_MANUALPB1, 
	ManualPB2:= OP10B_O_HORZ_MANUALPB2, 
	AutoCmd1:= OP10B_O_HORZ_AUTOCMD1, 
	AutoCmd2:= OP10B_O_HORZ_AUTOCMD2, 
	OperationEnable:= OperationEnable, 
	SafeHome:=, 
	SafeWork:=, 
	Pulse_1Sec:= Pulse_Block.Q1Hz, 
	BlinkingBit:= , 
	TimeOut1:= 5, 
	TimeOut2:= 5, 
	TimeOut3:= 5,
	HOMING_STRT:= (OP10B_HME_STP_NO= 15),
	HME_DLY:= 100,
	HME_DN_NO:= OP10B_HME_15_20,	
	HME_CYL_2:=TRUE ,
	HME_CYL_3:=TRUE , 
	Solenoid1=> O10B_ORING_HORZ_CYL_REV_Q1060_6, 
	Solenoid2=> O10B_ORING_HORZ_CYL_FWD_Q1060_7, 
	AlarmSensor1=> OP10B_HORZ_CYL_A1, 
	AlarmSensor2=> OP10B_HORZ_CYL_A2, 
	AlarmSolenoid1=> OP10B_HORZ_CYL_A3, 
	AlarmSolenoid2=> OP10B_HORZ_CYL_A4, 
	AllSignal=> OP10B_HORZ_CYL_A5, 
	AlarmPresent=> OP10B_CYLINDER_ERR.0, 
	Position1=> , 
	Position2=> , 
	HomeSensorBlink=> , 
	WorkSensorBlink=> ,	
	Status:= OP10B_HORZ_CYL_STUS,
	HMENG_RESULT := OP10B_HME_STP_NO);
	

// OP10B_VERT_CYLINDER_SAFE_WRK/HME
OP10B_VERT_CYL.SafeHome				:= OP10B_HORZ_CYL.Sensor1 OR OP10B_HORZ_CYL.Sensor2;
OP10B_VERT_CYL.SafeWork				:= (OP10B_HORZ_CYL.Sensor1 OR OP10B_HORZ_CYL.Sensor2) AND OP10B_DEGREE_CYL.Sensor1;
	
OP10B_VERT_CYL(
	Auto:= OP10B_AUTO_RUNNING OR OP10B_STEP_RUNNING OR OP10B_CYL_PNP_CHECK , 
	Manual:= OP10B_MANUAL_SELECTED,
	HOMING_RUNNING:= OP10B_START_HOMNG, 
	ErrorActive:= OP10B_ERR, 
	ResetPB:= Servo_Reset, 
	Sensor1:= I10B_ORING_VERT_CYL_UP_I1031_4, 
	Sensor2:= I10B_ORING_VERT_CYL_DWN_I1031_5, 								(*OP10B_VERT_CYL_FUNTIONAL_BLOCK*)
	ManualPB1:= OP10B_O_VERT_MANUALPB1, 
	ManualPB2:= OP10B_O_VERT_MANUALPB2, 
	AutoCmd1:= OP10B_O_VERT_AUTOCMD1, 
	AutoCmd2:= OP10B_O_VERT_AUTOCMD2, 
	OperationEnable:= OperationEnable, 
	SafeHome:= , 
	SafeWork:= , 
	Pulse_1Sec:= Pulse_Block.Q1Hz, 
	BlinkingBit:= , 
	TimeOut1:= 5, 
	TimeOut2:= 5, 
	TimeOut3:= 5,
	HOMING_STRT:= (OP10B_HME_STP_NO= 20),
	HME_DLY:= 100,
	HME_DN_NO:= OP10B_HME_20_25,
	HME_CYL_2:=TRUE ,
	HME_CYL_3:=TRUE , 
	Solenoid1=> O10B_ORING_VERT_CYL_UP_Q1061_0, 
	Solenoid2=> O10B_ORING_VERT_CYL_DWN_Q1061_1, 
	AlarmSensor1=> OP10B_VERT_CYL_A1, 
	AlarmSensor2=> OP10B_VERT_CYL_A2, 
	AlarmSolenoid1=> OP10B_VERT_CYL_A3, 
	AlarmSolenoid2=> OP10B_VERT_CYL_A4, 
	AllSignal=> OP10B_VERT_CYL_A5, 
	AlarmPresent=> OP10B_CYLINDER_ERR.1, 
	Position1=> , 
	Position2=> , 
	HomeSensorBlink=> , 
	WorkSensorBlink=> ,
	Status:= OP10B_VERT_CYL_STUS,
	HMENG_RESULT := OP10B_HME_STP_NO);

// OP10B_DEGREE_CYLINDER_SAFE_WRK/HME	
OP10B_DEGREE_CYL.SafeHome				:= OP10B_HORZ_CYL.Sensor1 AND OP10B_VERT_CYL.Sensor1;
OP10B_DEGREE_CYL.SafeWork				:= OP10B_HORZ_CYL.Sensor1 AND OP10B_VERT_CYL.Sensor1; 	
	
OP10B_DEGREE_CYL(
	Auto:= OP10B_AUTO_RUNNING OR OP10B_STEP_RUNNING OR OP10B_CYL_PNP_CHECK , 
	Manual:= OP10B_MANUAL_SELECTED,
	HOMING_RUNNING:= OP10B_START_HOMNG, 
	ErrorActive:= OP10B_ERR, 
	ResetPB:= Servo_Reset, 
	Sensor1:= I10B_ORING_ROTRY_CYL_O_DEG_I1031_0, 							(*OP10B_DEGREE_CYL_FUNTIONAL_BLCK*)
	Sensor2:= I10B_ORING_ROTRY_CYL_180_DEG_I1031_1, 
	ManualPB1:= OP10B_O_0DEGRE_MANUALPB1, 
	ManualPB2:= OP10B_O_180DEGRE_MANUALPB2, 
	AutoCmd1:= OP10B_O_0DEGRE_AUTOCMD1, 
	AutoCmd2:= OP10B_O_180DEGRE_AUTOCMD2, 
	OperationEnable:= OperationEnable, 
	SafeHome:=, 
	SafeWork:=, 
	Pulse_1Sec:= Pulse_Block.Q1Hz, 
	BlinkingBit:= , 
	TimeOut1:= 5, 
	TimeOut2:= 5, 
	TimeOut3:= 5,
	HOMING_STRT:= (OP10B_HME_STP_NO= 25),
	HME_DLY:= 100,
	HME_DN_NO:=  OP10B_HME_25_30,
	HME_CYL_2:=TRUE ,
	HME_CYL_3:=TRUE , 
	Solenoid1=> O10B_ORING_ROTRY_CYL_O_DEG_Q1060_4, 
	Solenoid2=> O10B_ORING_ROTRY_CYL_180_DEG_Q1060_5, 
	AlarmSensor1=> OP10B_DEGREE_CYL_A1, 
	AlarmSensor2=> OP10B_DEGREE_CYL_A2, 
	AlarmSolenoid1=> OP10B_DEGREE_CYL_A3, 
	AlarmSolenoid2=> OP10B_DEGREE_CYL_A4, 
	AllSignal=> OP10B_DEGREE_CYL_A5, 
	AlarmPresent=> OP10B_CYLINDER_ERR.2, 
	Position1=> , 
	Position2=> , 
	HomeSensorBlink=> , 
	WorkSensorBlink=> ,	
	Status:= OP10B_DEGREE_CYL_STUS,
	HMENG_RESULT := OP10B_HME_STP_NO);
// OP10B_LH_GRIPPER_CYLINDER_SAFE_WRK/HME	
OP10B_LH_GRP.SafeHome						:= OP10B_LH_PUSH.Sensor1;
OP10B_LH_GRP.SafeWork						:= OP10B_LH_PUSH.Sensor1;

OP10B_LH_GRP(
	Auto:= OP10B_AUTO_RUNNING OR OP10B_STEP_RUNNING OR OP10B_CYL_PNP_CHECK , 
	Manual:= OP10B_MANUAL_SELECTED,
	HOMING_RUNNING:= OP10B_START_HOMNG, 
	ErrorActive:= OP10B_ERR, 
	ResetPB:= Servo_Reset, 
	Sensor1:= I10B_ORING_LH_GRPR_CLSE_I1030_2, 								(*OP10B_LH_GRIPPER_FUNCATIONAL_BLOCK*)
	Sensor2:= I10B_ORING_LH_GRPR_OPN_I1030_3, 
	ManualPB1:=OP10B_MANUAL_SELECTED AND NOT OP10B_M_O_LHGRIP_ONOFF , 
	ManualPB2:=OP10B_MANUAL_SELECTED AND OP10B_M_O_LHGRIP_ONOFF, 
	AutoCmd1:=OP10B_LH_GRP.AUTO AND NOT OP10B_A_O_LHGRIP_ONOFF, 
	AutoCmd2:=OP10B_LH_GRP.AUTO AND OP10B_A_O_LHGRIP_ONOFF, 
	OperationEnable:= OperationEnable, 
	SafeHome:=, 
	SafeWork:=, 
	Pulse_1Sec:= Pulse_Block.Q1Hz, 
	BlinkingBit:= , 
	TimeOut1:= 5, 
	TimeOut2:= 5, 
	TimeOut3:= 5,
	HOMING_STRT:= (OP10B_HME_STP_NO= 5),
	HME_DLY:= 100,
	HME_DN_NO:= OP10B_HME_5_10,
	HME_CYL_2:=OP10B_RH_GRP.Sensor1,
	HME_CYL_3:=TRUE , 
	Solenoid1=> , 
	Solenoid2=> O10B_ORING_LH_GRPR_CLSE_OPN_Q1060_0, 
	AlarmSensor1=> OP10B_LH_GRP_A1, 
	AlarmSensor2=> OP10B_LH_GRP_A2, 
	AlarmSolenoid1=> OP10B_LH_GRP_A3, 
	AlarmSolenoid2=> OP10B_LH_GRP_A4, 
	AllSignal=> OP10B_LH_GRP_A5, 
	AlarmPresent=> OP10B_CYLINDER_ERR.3, 
	Position1=> , 
	Position2=> , 
	HomeSensorBlink=> , 
	WorkSensorBlink=> ,	
	Status:= OP10B_LH_GRP_STATS,
	HMENG_RESULT := OP10B_HME_STP_NO);

// OP10B_RH_GRIPPER_CYLINDER_SAFE_WRK/HME	
OP10B_RH_GRP.SafeHome						:= OP10B_RH_PUSH.Sensor1;
OP10B_RH_GRP.SafeWork						:= OP10B_RH_PUSH.Sensor1;				// CHANGE THE INPUT AS FALSE

OP10B_RH_GRP(
	Auto:= OP10B_AUTO_RUNNING OR OP10B_STEP_RUNNING OR OP10B_CYL_PNP_CHECK  , 
	Manual:= OP10B_MANUAL_SELECTED,
	HOMING_RUNNING:= OP10B_START_HOMNG, 
	ErrorActive:= OP10B_ERR, 
	ResetPB:= Servo_Reset, 
	Sensor1:=I10B_ORING_RH_GRPR_CLSE_I1030_6 , 
	Sensor2:=I10B_ORING_RH_GRPR_OPN_I1030_5 , 
	ManualPB1:=OP10B_MANUAL_SELECTED AND NOT OP10B_M_O_RHGRIP_ONOFF, 
	ManualPB2:=OP10B_MANUAL_SELECTED AND OP10B_M_O_RHGRIP_ONOFF, 									(*OP10B_RH_GRIPPER_CYLINDER*)
	AutoCmd1:=OP10B_RH_GRP.AUTO AND NOT OP10B_A_O_RHGRIP_ONOFF, 
	AutoCmd2:=OP10B_RH_GRP.AUTO AND OP10B_A_O_RHGRIP_ONOFF, 
	OperationEnable:= OperationEnable, 
	SafeHome:= , 
	SafeWork:= , 
	Pulse_1Sec:= Pulse_Block.Q1Hz, 
	BlinkingBit:= , 
	TimeOut1:= 5, 
	TimeOut2:= 5, 
	TimeOut3:= 5,
	HOMING_STRT:= (OP10B_HME_STP_NO= 5),
	HME_DLY:= 100,
	HME_DN_NO:= ,
	HME_CYL_2:=TRUE ,
	HME_CYL_3:=TRUE , 
	Solenoid1=> , 
	Solenoid2=> O10B_ORING_RH_GRPR_CLSE_OPN_Q1060_2, 
	AlarmSensor1=> OP10B_RH_GRP_A1, 
	AlarmSensor2=> OP10B_RH_GRP_A2, 
	AlarmSolenoid1=> OP10B_RH_GRP_A3, 
	AlarmSolenoid2=> OP10B_RH_GRP_A4, 
	AllSignal=> OP10B_RH_GRP_A5, 
	AlarmPresent=> OP10B_CYLINDER_ERR.4, 
	Position1=> , 
	Position2=> , 
	HomeSensorBlink=> , 
	WorkSensorBlink=> ,	
	Status:= OP10B_RH_GRP_STUS,
	HMENG_RESULT := OP10B_PARLLEL);

// OP10B_LH_PUSH_CYLINDER_SAFE_WRK/HME
OP10B_LH_PUSH.SafeHome						:=OP10B_LH_GRP.Sensor2 ;
OP10B_LH_PUSH.SafeWork						:=OP10B_LH_GRP.Sensor2 ;
	
OP10B_LH_PUSH(
	Auto:= OP10B_AUTO_RUNNING OR OP10B_STEP_RUNNING OR OP10B_CYL_PNP_CHECK , 
	Manual:= OP10B_MANUAL_SELECTED,
	HOMING_RUNNING:= OP10B_START_HOMNG, 
	ErrorActive:= OP10B_ERR, 
	ResetPB:= Servo_Reset, 
	Sensor1:= NOT I10B_ORING_LH_PUSHR_CYL_REV_I1030_4, 										(*OP10B_LH_PUSHING_CYLINDER*)
	Sensor2:= I10B_ORING_LH_PUSHR_CYL_REV_I1030_4, 
	ManualPB1:=OP10B_MANUAL_SELECTED AND NOT OP10B_M_O_LHPUSH_CYL, 
	ManualPB2:=OP10B_MANUAL_SELECTED AND OP10B_M_O_LHPUSH_CYL, 
	AutoCmd1:= OP10B_LH_PUSH.AUTO AND NOT OP10B_A_O_LHPUSH_CYL, 
	AutoCmd2:= OP10B_LH_PUSH.AUTO AND OP10B_A_O_LHPUSH_CYL, 
	OperationEnable:= OperationEnable, 
	SafeHome:= 1, 
	SafeWork:= 1, 
	Pulse_1Sec:= Pulse_Block.Q1Hz, 
	BlinkingBit:= , 
	TimeOut1:= 5, 
	TimeOut2:= 5, 
	TimeOut3:= 5,
	HOMING_STRT:= (OP10B_HME_STP_NO= 1),
	HME_DLY:= 100,
	HME_DN_NO:= OP10B_HME_1_5,
	HME_CYL_2:=OP10B_RH_PUSH.Sensor1,
	HME_CYL_3:=TRUE , 
	Solenoid1=> , 
	Solenoid2=> O10B_ORING_LH_PUSHR_CYL_REV_FWD_Q1060_1, 
	AlarmSensor1=> OP10B_LH_PUSH_A1, 
	AlarmSensor2=> OP10B_LH_PUSH_A2, 
	AlarmSolenoid1=> OP10B_LH_PUSH_A3, 
	AlarmSolenoid2=> OP10B_LH_PUSH_A4, 
	AllSignal=> OP10B_LH_PUSH_A5, 
	AlarmPresent=> OP10B_CYLINDER_ERR.5, 
	Position1=> , 
	Position2=> , 
	HomeSensorBlink=> , 
	WorkSensorBlink=> ,
	Status:= OP10B_LH_PUSH_STUS,
	HMENG_RESULT := OP10B_HME_STP_NO);

// OP10B_LH_PUSH_CYLINDER_SAFE_WRK/HME
OP10B_RH_PUSH.SafeHome						:= OP10B_RH_GRP.Sensor2 ;
OP10B_RH_PUSH.SafeWork						:= OP10B_RH_GRP.Sensor2 ;

OP10B_RH_PUSH(
	Auto:= OP10B_AUTO_RUNNING OR OP10B_STEP_RUNNING OR OP10B_CYL_PNP_CHECK , 
	Manual:= OP10B_MANUAL_SELECTED,
	HOMING_RUNNING:= OP10B_START_HOMNG, 
	ErrorActive:= OP10B_ERR, 								(*OP10B_RH _ PUSHING CYL_FUNTIONAL_BLCK*)
	ResetPB:= Servo_Reset, 
	Sensor1:= NOT I10B_ORING_RH_PUSHR_CYL_REV_I1030_7, 
	Sensor2:=I10B_ORING_RH_PUSHR_CYL_REV_I1030_7 , 
	ManualPB1:=OP10B_MANUAL_SELECTED AND NOT OP10B_M_O_RHPUSH_CYL, 
	ManualPB2:=OP10B_MANUAL_SELECTED AND OP10B_M_O_RHPUSH_CYL, 
	AutoCmd1:=OP10B_RH_PUSH.Auto AND NOT OP10B_A_O_RHPUSH_CYL, 
	AutoCmd2:=OP10B_RH_PUSH.Auto AND OP10B_A_O_RHPUSH_CYL, 
	OperationEnable:= OperationEnable, 
	SafeHome:= 1, 
	SafeWork:= 1, 
	Pulse_1Sec:= Pulse_Block.Q1Hz, 
	BlinkingBit:= , 
	TimeOut1:= 5, 
	TimeOut2:= 5, 
	TimeOut3:= 5,
	HOMING_STRT:= (OP10B_HME_STP_NO=1),
	HME_DLY:= ,
	HME_DN_NO:= ,	
	HME_CYL_2:=TRUE ,
	HME_CYL_3:=TRUE , 
	Solenoid1=> , 
	Solenoid2=>O10B_ORING_RH_PUSHR_CYL_REV_FWD_Q1060_3 , 
	AlarmSensor1=> OP10B_RH_PUSH_A1, 
	AlarmSensor2=> OP10B_RH_PUSH_A2, 
	AlarmSolenoid1=> OP10B_RH_PUSH_A3, 
	AlarmSolenoid2=> OP10B_RH_PUSH_A4, 
	AllSignal=> OP10B_RH_PUSH_A5, 
	AlarmPresent=> OP10B_CYLINDER_ERR.6, 
	Position1=> , 
	Position2=> , 
	HomeSensorBlink=> , 
	WorkSensorBlink=> ,	
	Status:= OP10B_RH_PUSH_STUS,
	HMENG_RESULT := OP10B_PARLLEL);

// OP10B_LH_REJ_CYLINDER_SAFE_WRK/HME
//OP10B_LH_REJ.SafeHome						:= TRUE;
//OP10B_LH_REJ.SafeWork						:= TRUE;

OP10B_LH_REJ(
	Auto:= OP10B_AUTO_RUNNING OR OP10B_STEP_RUNNING OR OP10B_CYL_PNP_CHECK, 
	Manual:= OP10B_MANUAL_SELECTED,
	HOMING_RUNNING:= OP10B_START_HOMNG, 
	ErrorActive:= OP10B_ERR, 								(*OP10B_RH _ PUSHING CYL_FUNTIONAL_BLCK*)
	ResetPB:= Servo_Reset, 
	Sensor1:=I10B_LH_FIRTRE_ORING_REJ_CYL_REV_I1031_6, 											 
	Sensor2:=I10B_LH_FIRTRE_ORING_REJ_CYL_FWD_I1031_7,                                              
	ManualPB1:= OP10B_M_LH_REJ_HOME,                        
	ManualPB2:= OP10B_M_LH_REJ_WRK,
	AutoCmd1:= OP10B_A_LH_REJ_HOME,                                              
	AutoCmd2:= OP10B_A_LH_REJ_WRK,                                              
	OperationEnable:= OperationEnable, 
	SafeHome:= 1, 
	SafeWork:= 1, 
	Pulse_1Sec:= Pulse_Block.Q1Hz, 
	BlinkingBit:= , 
	TimeOut1:= 5, 
	TimeOut2:= 5, 
	TimeOut3:= 5,
	HOMING_STRT:= (OP10B_HME_STP_NO=1),
	HME_DLY:= ,
	HME_DN_NO:= ,
	HME_CYL_2:=TRUE ,
	HME_CYL_3:=TRUE , 
	Solenoid1=>O10B_LH_FIRTRE_ORING_REJ_CYL_REV_Q1061_2 , 
	Solenoid2=> O10B_LH_FIRTRE_ORING_REJ_CYL_FWD_Q1061_3, 
	AlarmSensor1=> OP10B_LH_REJ_A1,	
	AlarmSensor2=>OP10B_LH_REJ_A2,	
	AlarmSolenoid1=>OP10B_LH_REJ_A3,	
	AlarmSolenoid2=>OP10B_LH_REJ_A4,	
	AllSignal=> OP10B_LH_REJ_A5,	
	AlarmPresent=> OP10B_CYLINDER_ERR.7, 
	Position1=> , 
	Position2=> , 
	HomeSensorBlink=> , 
	WorkSensorBlink=> ,	
	Status:= OP10B_RH_PUSH_STUS,
	HMENG_RESULT := OP10B_PARLLEL);	
	
// OP10B_RH_REJ_CYLINDER_SAFE_WRK/HME
//OP10B_RH_REJ.SafeHome						:= TRUE;
//OP10B_RH_REJ.SafeWork						:= TRUE;

OP10B_RH_REJ(
	Auto:= OP10B_AUTO_RUNNING OR OP10B_STEP_RUNNING OR OP10B_CYL_PNP_CHECK, 
	Manual:= OP10B_MANUAL_SELECTED,
	HOMING_RUNNING:= OP10B_START_HOMNG, 
	ErrorActive:= OP10B_ERR, 								(*OP10B_RH _ PUSHING CYL_FUNTIONAL_BLCK*)
	ResetPB:= Servo_Reset, 
	Sensor1:= I10B_RH_FIRTRE_ORING_REJ_CYL_REV_I1040_0 , 
	Sensor2:= I10B_RH_FIRTRE_ORING_REJ_CYL_FWD_I1040_1 , 
	ManualPB1:= OP10B_M_RH_REJ_HOME,		
	ManualPB2:= OP10B_M_RH_REJ_WRK,	  
	AutoCmd1:= OP10B_A_RH_REJ_HOME, 
	AutoCmd2:= OP10B_A_RH_REJ_WRK, 
	OperationEnable:= OperationEnable, 
	SafeHome:= 1, 
	SafeWork:= 1, 
	Pulse_1Sec:= Pulse_Block.Q1Hz, 
	BlinkingBit:= , 
	TimeOut1:= 5, 
	TimeOut2:= 5, 
	TimeOut3:= 5,
	HOMING_STRT:= (OP10B_HME_STP_NO=1),
	HME_DLY:= ,
	HME_DN_NO:= ,
	HME_CYL_2:=TRUE ,
	HME_CYL_3:=TRUE , 
	Solenoid1=>O10B_RH_FIRTRE_ORING_REJ_CYL_REV_Q1061_4 , 
	Solenoid2=>O10B_RH_FIRTRE_ORING_REJ_CYL_FWD_Q1061_5 , 
	AlarmSensor1=> OP10B_RH_REJ_A1,	
	AlarmSensor2=> OP10B_RH_REJ_A2,	
	AlarmSolenoid1=> OP10B_RH_REJ_A3,	
	AlarmSolenoid2=>OP10B_RH_REJ_A4,	
	AllSignal=>OP10B_RH_REJ_A5,	
	AlarmPresent=> OP10B_CYLINDER_ERR.8, 
	Position1=> , 
	Position2=> , 
	HomeSensorBlink=> , 
	WorkSensorBlink=> ,	
	Status:= OP10B_RH_PUSH_STUS,
	HMENG_RESULT := OP10B_PARLLEL);	

	
////////////////////////////////////////OP10 SINGULATING GRIPPER/////////////////////////////


OP10_BDY_SING_FRT(
	Auto:= (OP10A_AUTO_RUNNING OR  OP10A_STEP_RUNNING )OR (OP10B_AUTO_RUNNING OR OP10B_STEP_RUNNING) OR CHECK, 
	Manual:= OP10B_MANUAL_SELECTED AND OP10A_MANUAL_SELECTED AND NOT CHECK,
	HOMING_RUNNING:= (OP10A_START_HOMNG OR OP10B_START_HOMNG), 
	ErrorActive:= (OP10B_ERR AND NOT OP10B_BYPASS) OR (OP10A_ERR AND NOT OP10A_BYPASS), 								(*OP10B_RH _ PUSHING CYL_FUNTIONAL_BLCK*)
	ResetPB:= Servo_Reset, 
	Sensor1:= I10A_BDY_SING_CYL_CLSE_I1020_2,  
	Sensor2:= I10A_BDY_SING_CYL_OPN_I1020_3,  
	ManualPB1:=OP10_FRT_BDY_SING_HME,											
	ManualPB2:=OP10_FRT_BDY_SING_WRK,	                                    	
	AutoCmd1:= OP10_A_FRT_BDY_SING_HME,                                        	
	AutoCmd2:= OP10_A_FRT_BDY_SING_WRK,                                        	
	OperationEnable:= OperationEnable, 
	SafeHome:= 1, 
	SafeWork:= 1, 
	Pulse_1Sec:= Pulse_Block.Q1Hz, 
	BlinkingBit:= , 
	TimeOut1:= 5, 
	TimeOut2:= 5, 
	TimeOut3:= 5,
	HOMING_STRT:= OP10_FRT_CYL_INITZAL,
	HME_DLY:= ,
	HME_DN_NO:= ,
	HME_CYL_2:=TRUE ,
	HME_CYL_3:=TRUE , 
	Solenoid1=>O10A_BDY_SING_CYL_CLSE_Q1051_6, 
	Solenoid2=>O10A_BDY_SING_CYL_OPN_Q1051_7,  
	AlarmSensor1=>OP10_BDY_SING_FRT_A1,	
	AlarmSensor2=>OP10_BDY_SING_FRT_A2,	
	AlarmSolenoid1=>OP10_BDY_SING_FRT_A3,	
	AlarmSolenoid2=>OP10_BDY_SING_FRT_A4,	
	AllSignal=>OP10_BDY_SING_FRT_A5,	
	AlarmPresent=> OP10A_CYLINDER_ERR.9, 
	Position1=> , 
	Position2=> , 
	HomeSensorBlink=> , 
	WorkSensorBlink=> ,	
	Status:= OP10_BDY_SING_FRT_STATUS,
	HMENG_RESULT := OP10B_PARLLEL);


OP10_BDY_SING_SEC(
	Auto:= (OP10A_AUTO_RUNNING OR  OP10A_STEP_RUNNING )OR (OP10B_AUTO_RUNNING OR OP10B_STEP_RUNNING) OR CHECK, 
	Manual:= OP10B_MANUAL_SELECTED AND OP10A_MANUAL_SELECTED AND NOT CHECK,
	HOMING_RUNNING:= (OP10A_START_HOMNG OR OP10B_START_HOMNG), 
	ErrorActive:= (OP10B_ERR AND NOT OP10B_BYPASS) OR (OP10A_ERR AND NOT OP10A_BYPASS), 								(*OP10B_RH _ PUSHING CYL_FUNTIONAL_BLCK*)
	ResetPB:= Servo_Reset, 
	Sensor1:= I10B_BDY_SING_CYL_CLSE_I1040_2,   
	Sensor2:= I10B_BDY_SING_CYL_OPN_I1040_3,   
	ManualPB1:=OP10_SEC_BDY_SING_HME,		
	ManualPB2:=OP10_SEC_BDY_SING_WRK,	  
	AutoCmd1:= OP10_A_SEC_BDY_SING_HME, 
	AutoCmd2:= OP10_A_SEC_BDY_SING_WRK, 
	OperationEnable:= OperationEnable, 
	SafeHome:= 1, 
	SafeWork:= 1, 
	Pulse_1Sec:= Pulse_Block.Q1Hz, 
	BlinkingBit:= , 
	TimeOut1:= 5, 
	TimeOut2:= 5, 
	TimeOut3:= 5,
	HOMING_STRT:=OP10_SEC_CYL_INITZAL,
	HME_DLY:= ,
	HME_DN_NO:= ,
	HME_CYL_2:=TRUE ,
	HME_CYL_3:=TRUE , 
	Solenoid1=> O10B_BDY_SING_CYL_CLSE_Q1061_6,  
	Solenoid2=> O10B_BDY_SING_CYL_OPN_Q1061_7,   
	AlarmSensor1=> , 
	AlarmSensor2=> , 
	AlarmSolenoid1=>, 
	AlarmSolenoid2=> , 
	AllSignal=> , 
	AlarmPresent=> OP10A_CYLINDER_ERR.10, 
	Position1=> , 
	Position2=> , 
	HomeSensorBlink=> , 
	WorkSensorBlink=> ,	
	HMENG_RESULT=>  , 
	Status:= OP10_BDY_SING_SEC_STATUS,
	HMENG_RESULT := OP10B_PARLLEL);

END_PROGRAM

(* stored: Version 1.1.0.1, ProductVersion 3.1.4024.11
   POU OP10_MANUAL: Id {9e7f684a-f156-4b15-9ac9-b8d545a62920}, SpecialFunc None *)
